(*			
	EVERDE sp. z o.o.
	Rafał Osajda		08.08.2025		TC 4024.66
	Interfejs do wyciągania z SPM przez HMI danych do wyświetlania - dla ramki statystyki
*)
INTERFACE ITF_SPM_HMI_05_Lacznik EXTENDS  B_Baza.ITF_ZrodloIdentyfikacji

END_INTERFACE

(* stored: Version 1.1.0.1
   Itf ITF_SPM_HMI_05_Lacznik: Id {848bd6cd-ead0-09b3-018d-ba5afd466816} *)
